FUNCTION_BLOCK CmdSludgeDischargeSLB_HMI (* Service Interface Function Block Type *)
  (* Standard: 61499-2 *)
  (* Version 2.0, 10/1/2026, Schneider Electric, Rev2 - Cmin (velocidade minima por bomba, evento PUMP_MIN_PAR); valores padrao; template *)
  PACKAGE SE.Nereda;
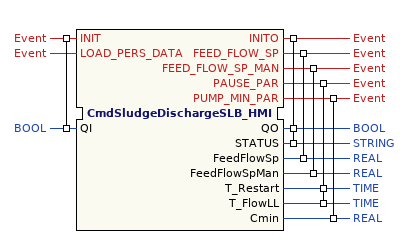
  EVENT_INPUT
    INIT WITH QI;
    LOAD_PERS_DATA;
  END_EVENT
  EVENT_OUTPUT
    INITO WITH QO, STATUS;
    FEED_FLOW_SP WITH FeedFlowSp;
    FEED_FLOW_SP_MAN WITH FeedFlowSpMan;
    PAUSE_PAR WITH T_Restart, T_FlowLL; (* Parametros da pausa da descarga de lodo *)
    PUMP_MIN_PAR WITH Cmin; (* Velocidade minima das bombas *)
  END_EVENT
  VAR_INPUT
    QI : BOOL;
  END_VAR
  VAR_OUTPUT
    QO : BOOL; (* Event Output Qualifier *)
    STATUS : STRING; (* Service Status *)
    FeedFlowSp : REAL;
    FeedFlowSpMan : REAL;
    T_Restart : TIME; (* Pausa: tempo para retomar apos a causa (nivel L / vazao LL) sair *)
    T_FlowLL : TIME; (* Vazao LL do 49FT0004 com bomba rodando por este tempo = pausa (0 = desabilitado) *)
    Cmin : REAL; (* Velocidade minima de cada bomba em servico [% velocidade] *)
  END_VAR
  SERVICE /
    SEQUENCE 
    END_SEQUENCE
  END_SERVICE
END_FUNCTION_BLOCK
